FUNCTION_BLOCK FB_TrajectoryGenerator
VAR_INPUT
END_VAR
VAR_OUTPUT
END_VAR
VAR
	eCondition : eConditionCheck;
	
	//ErrorBits
	bNoConnectionToXMC1 : BIT;
	bNoConnectionToXMC2 : BIT;
	bNoConnectionToXMC3 : BIT;
	bNoConnectionToXMC4 : BIT;
END_VAR

PROPERTY PUBLIC getErrorBits : UDINT
GET



getErrorBits.0 := bNoConnectionToXMC1;
getErrorBits.1 := bNoConnectionToXMC2;
getErrorBits.2 := bNoConnectionToXMC3;
getErrorBits.3 := bNoConnectionToXMC4;
END_GET
END_PROPERTY

END_FUNCTION_BLOCK

(* stored: Version 1.1.0.1, ProductVersion 3.1.4024.12
   POU FB_TrajectoryGenerator: Id {0fe2a302-c596-4eee-ba7e-45869f82e2bc}, SpecialFunc None
   Property getErrorBits: Id {2190d3fb-f308-4551-a1c4-7e82ba23d84f}
   Get Get: Id {54f29ea6-985f-45e3-bb86-9d768df60d77} *)
